{attribute 'reflection'} 
FUNCTION_BLOCK ABSTRACT FB_Base EXTENDS  FB_SkillHandler  IMPLEMENTS ITF_0_BaseComponent
VAR_INPUT
END_VAR
VAR_OUTPUT
END_VAR
VAR
	{attribute 'instance-path'} 
    {attribute 'noinit'} 
    sPath : STRING; 
	{attribute 'instance-name'}
	{attribute 'noinit'} 
	sInstanceName: STRING;
	_autoboot: BOOL:=TRUE;		//If True, StateMachine trys automatic to reach State "ACTIV" otherwise each transition must be called manually
	
	transitionresult: eResult;
	_state: eState :=eState.Unconfigured;
	

	dummy: INT;
END_VAR

StateMachine();

{warning 'Add method implementation '}
METHOD M_activate : BOOL
IF P_State=eState.Inactive THEN
	P_State:=eState.Activating;
END_IF
END_METHOD

{warning 'Add method implementation '}
METHOD M_cleanup : BOOL
IF P_State=eState.Inactive THEN
	P_State:=eState.CleaningUp;
END_IF
END_METHOD

{warning 'Add method implementation '}
METHOD M_configure : BOOL
IF P_State=eState.Unconfigured THEN
	P_State:=eState.Configuring;
END_IF
END_METHOD

{warning 'Add method implementation '}
METHOD M_deactivate : BOOL
IF P_State=eState.Active THEN
	P_State:=eState.Deactivating;
END_IF
END_METHOD

{warning 'Add method implementation '}
METHOD M_destroy : BOOL
IF P_State=eState.Finalized THEN
	P_State:=eState.Unconfigured;
END_IF
END_METHOD

{warning 'Add method implementation '}
METHOD M_shutdown : BOOL
IF P_State=eState.Inactive OR P_State=eState.Unconfigured OR P_State=eState.Active THEN
	P_State:=eState.ShuttingDown;
END_IF
END_METHOD

METHOD onActivate : BOOL
// ---- Init ----
transitionresult:=eResult.None;



// ---- Change ----



// ---- Check ----
transitionresult := eResult.SUCCESS;


// ---- Change State ----
IF transitionresult= eResult.SUCCESS THEN
	P_State:=eState.Active;
ELSIF transitionresult= eResult.FAILURE THEN
	P_State:=eState.Inactive;
ELSIF transitionresult= eResult.ERROR THEN
	P_State:=eState.ErrorProcessing;
ELSE
	ADSLOGSTR(ADSLOG_MSGTYPE_WARN,'Transitionresult from onActivate is None','');
END_IF
END_METHOD

METHOD onCleanup : BOOL
// ---- Init ----
transitionresult:=eResult.None;



// ---- Change ----



// ---- Check ----
transitionresult := eResult.SUCCESS;


// ---- Change State ----
IF transitionresult= eResult.SUCCESS THEN
	P_State:=eState.Unconfigured;
ELSIF transitionresult= eResult.FAILURE THEN
	ADSLOGSTR(ADSLOG_MSGTYPE_WARN,'Transitionresult from onCleanup is FAILURE ','');
ELSIF transitionresult= eResult.ERROR THEN
	P_State:=eState.ErrorProcessing;
ELSE
	ADSLOGSTR(ADSLOG_MSGTYPE_WARN,'Transitionresult from onCleanup is NONE','');
END_IF
END_METHOD

METHOD onConfigure : BOOL
// ---- Init ----
transitionresult:=eResult.None;



// ---- Change ----




// ---- Check ----
transitionresult := eResult.SUCCESS;


// ---- Change State ----
IF transitionresult= eResult.SUCCESS THEN
	P_State:=eState.Inactive;
ELSIF transitionresult= eResult.FAILURE THEN
	P_State:=eState.Unconfigured;
ELSIF transitionresult= eResult.ERROR THEN
	P_State:=eState.ErrorProcessing;
ELSE
	ADSLOGSTR(ADSLOG_MSGTYPE_WARN,'Transitionresult from onConfigure is None','');
END_IF
END_METHOD

METHOD onDeactivate : BOOL
// ---- Init ----
transitionresult:=eResult.None;



// ---- Change ----



// ---- Check ----
transitionresult := eResult.SUCCESS;


// ---- Change State ----
IF transitionresult= eResult.SUCCESS THEN
	P_State:=eState.Inactive;
ELSIF transitionresult= eResult.FAILURE THEN
	ADSLOGSTR(ADSLOG_MSGTYPE_WARN,'Transitionresult from onDeactivate is FAILURE','');
ELSIF transitionresult= eResult.ERROR THEN
	P_State:=eState.ErrorProcessing;
ELSE
	ADSLOGSTR(ADSLOG_MSGTYPE_WARN,'Transitionresult from onDeactivate is None','');
END_IF
END_METHOD

METHOD onError : BOOL
// ---- Init ----
transitionresult:=eResult.None;



// ---- Change ----




// ---- Check ----
transitionresult := eResult.SUCCESS;


// ---- Change State ----
IF transitionresult= eResult.SUCCESS THEN
	P_State:=eState.Unconfigured;
ELSIF transitionresult= eResult.FAILURE THEN
	P_State:=eState.Finalized;
ELSIF transitionresult= eResult.ERROR THEN
	ADSLOGSTR(ADSLOG_MSGTYPE_WARN,'Transitionresult from onError is Error','');
ELSE
	ADSLOGSTR(ADSLOG_MSGTYPE_WARN,'Transitionresult from onError is None','');
END_IF
END_METHOD

METHOD onShutdown : BOOL
// ---- Init ----
transitionresult:=eResult.None;



// ---- Change ----



// ---- Check ----
transitionresult := eResult.SUCCESS;


// ---- Change State ----
IF transitionresult= eResult.SUCCESS THEN
	P_State:=eState.Finalized;
ELSIF transitionresult= eResult.FAILURE THEN
	ADSLOGSTR(ADSLOG_MSGTYPE_WARN,'Transitionresult from onShutdown is FAILURE','');
ELSIF transitionresult= eResult.ERROR THEN
	P_State:=eState.ErrorProcessing;
ELSE
	ADSLOGSTR(ADSLOG_MSGTYPE_WARN,'Transitionresult from onShutdown is None','');
END_IF
END_METHOD

PROPERTY P_AutoBoot : BOOL
GET
P_AutoBoot:=_autoboot;
END_GET
SET
_autoboot:=P_AutoBoot;
END_SET
END_PROPERTY

{warning 'Add property implementation'}
PROPERTY P_ID : UINT
GET
END_GET
SET
END_SET
END_PROPERTY

{warning 'Add property implementation'}
PROPERTY P_Name : STRING
GET


P_Name:=sInstanceName;
END_GET
END_PROPERTY

{warning 'Add property implementation'}
PROPERTY P_Path : STRING
GET
P_Path:=sPath;
END_GET
END_PROPERTY

{warning 'Add property implementation'}
PROPERTY P_State : eState
GET
P_State:=_state;
END_GET
SET
_state:=P_State;
END_SET
END_PROPERTY

METHOD StateMachine : eState
VAR_INPUT
END_VAR
CASE _state OF
	eState.Unconfigured:
		IF _autoboot THEN
			M_configure();
		END_IF
	eState.Inactive:		//IDLE
// 		IF _autoboot THEN
// 			M_activate();
// 		END_IF
	eState.Active:
		dummy:=1;
	eState.Finalized:
		M_destroy();
	
	
	//Transitions States
	eState.Configuring:
		onConfigure();
	eState.Activating:
		onActivate();
	eState.Deactivating:
		onDeactivate();
	eState.ErrorProcessing:
		onError();
	eState.CleaningUp:
		onCleanup();
	eState.ShuttingDown:
		onShutdown();
		
END_CASE
END_METHOD

END_FUNCTION_BLOCK

(* stored: Version 1.1.0.1, ProductVersion 3.1.4026.18
   POU FB_Base: Id {ccfcc891-ed7a-48a9-bb43-020f08aa1f30}, SpecialFunc None
   Folder StateControl: Id {bcaabc90-8311-4d61-b63c-66c13d25292f}
   Method M_activate: Id {8d29e9eb-3e7c-4311-8303-d07f52bcf283}
   Method M_cleanup: Id {c4819076-2442-41bd-8aa1-fe9bd8639fb5}
   Method M_configure: Id {e049feb0-d020-4b0d-9355-74a020722637}
   Method M_deactivate: Id {4dfdb93c-87ba-4697-9eee-0c2811499a1b}
   Method M_destroy: Id {84232af5-24cf-43e3-b44a-0f85cd0c58bf}
   Method M_shutdown: Id {a12b67df-13c4-4acd-81a2-259afa6359fe}
   Method onActivate: Id {9da44456-9079-48c4-a422-180073049c7f}
   Method onCleanup: Id {1cbf57cd-f144-4499-ac40-e58b878ddcfc}
   Method onConfigure: Id {c7df3a26-6fc2-40b8-b279-df837148749a}
   Method onDeactivate: Id {46dc1863-bc20-4aa6-822e-d746ed6280bd}
   Method onError: Id {c4fcde18-52a6-416e-9375-25c35d4fb566}
   Method onShutdown: Id {05a5db8e-a9c0-4764-9498-22b8037c7c75}
   Property P_AutoBoot: Id {44f3c7f4-dba0-4e5c-9aec-1d95215b519e}
   Get Get: Id {ee124298-bcc7-439c-9105-d90c42f3e44b}
   Set Set: Id {6e39cfd8-2d79-4d05-8c85-3f94875be35d}
   Property P_ID: Id {56e403f3-8552-4f82-8f86-af916d784dec}
   Get Get: Id {01362321-941b-405e-a5c3-370fadd50709}
   Set Set: Id {53535a56-c051-4863-b3cf-33275af6d47b}
   Property P_Name: Id {548614ea-6498-4c1d-a5ce-7f6dbb849726}
   Get Get: Id {9abd0c45-0dec-4466-a4b2-9f1564c8ba2e}
   Property P_Path: Id {459f7f21-cbfe-4701-91b3-a410fc19512e}
   Get Get: Id {2daa2808-fefd-47e5-b0e8-8c13e9ff4c08}
   Property P_State: Id {186f624f-e691-4cfe-9392-dd87366cedc2}
   Get Get: Id {8c20bc39-5e17-48de-81e9-f86cdcf5978c}
   Set Set: Id {f2b0cb44-bade-4a8a-80d6-a1f37ebc07e9}
   Method StateMachine: Id {2f358a4c-c272-4679-b042-e935cc28a3dc} *)
